(* PLC project  *)

FUNCTION MyFunction : BOOL
  VAR_INPUT
    Input1 : INT;
  END_VAR
  VAR_OUTPUT
    Output1 : DINT;
  END_VAR
  VAR
    Local1 : REAL := 0.0;
  END_VAR

            Output1 := Input1 * 2;
          
END_FUNCTION

FUNCTION_BLOCK MyFunctionBlock
  VAR_IN_OUT
    Counter : UDINT;
  END_VAR

            Counter := Counter + 1;
          
END_FUNCTION_BLOCK

PROGRAM MyProgram
  VAR_TEMP
    Temp : STRING;
  END_VAR

            Temp := 'Hello';
          
END_PROGRAM
